// Mitsubishi GX Works2 project: BookEX2_2 Conveyor   PLC: Q13UDV

TYPE cnvBlk : STRUCT
  PIDno : DINT;  (* Pid for ECS *)
  DestBlk : INT;  (* Dest Block *)
  Status : WORD;  (* control status *)
END_STRUCT END_TYPE

// global labels: Global
VAR_GLOBAL
  gCnvBuff : ARRAY [0..19] OF cnvBlk;  (* D100~  size:4x20 = 80 word *)
  gbBlkFinish : ARRAY [0..19] OF BOOL;
  gbBlkSen : ARRAY [0..19] OF BOOL;
  gbBlkSenOn : ARRAY [0..19] OF BOOL;
  gbBlkSenOff : ARRAY [0..19] OF BOOL;
  gbBlkUp : ARRAY [0..19] OF BOOL;
  gbBlkDw : ARRAY [0..19] OF BOOL;
  gbBlkTO : ARRAY [0..19] OF BOOL;
  gbBlkTrip : ARRAY [0..19] OF BOOL;
  gbBlkData : ARRAY [0..19] OF BOOL;
  gbBlkRun : ARRAY [0..19] OF BOOL;
  gbBlkRun2 : ARRAY [0..19] OF BOOL;
  gbBlkRunUp : ARRAY [0..19] OF BOOL;
  gbBlkRunDw : ARRAY [0..19] OF BOOL;
  gbBlkRunOk : ARRAY [0..19] OF BOOL;
  gbBlkRunOk2 : ARRAY [0..19] OF BOOL;
  gbBlkEnterOk : ARRAY [0..19] OF BOOL;
END_VAR
VAR_GLOBAL CONSTANT
  cOnTime : TIME := T#300ms;
END_VAR
VAR_GLOBAL
  swOPAuto : BOOL;
  swOPEmrg : BOOL;
  gbBlkColl : BOOL;
  swNormal : BOOL;
END_VAR
VAR_GLOBAL CONSTANT
  cMaxBlk : INT := 19;
END_VAR
VAR_GLOBAL
  gwTemp AT D100 : WORD;
END_VAR
VAR_GLOBAL CONSTANT
  cMaxTime : TIME := T#15s;
  cSimTime : TIME := T#5s;
END_VAR
VAR_GLOBAL
  man01 : BOOL;
  man02 : BOOL;
  man03 : BOOL;
  man04 : BOOL;
  man05 : BOOL;
  man06 : BOOL;
  man07 : BOOL;
  man08 : BOOL;
  man09 : BOOL;
  man10 : BOOL;
  man11 : BOOL;
  man02E : BOOL;
  man05E : BOOL;
  man09E : BOOL;
  man12 : BOOL;
  man13 : BOOL;
  man12E : BOOL;
  man02Up : BOOL;
  man02Dw : BOOL;
  man05Up : BOOL;
  man05Dw : BOOL;
  man09Up : BOOL;
  man09Dw : BOOL;
  man12Up : BOOL;
  man12Dw : BOOL;
END_VAR
VAR_GLOBAL CONSTANT
  cOffTime : TIME := T#300ms;
END_VAR
VAR_GLOBAL
  swJobCmd : BOOL;
  swJobDel : BOOL;
  xSen01 AT X120 : BOOL;
  xSen02 AT X121 : BOOL;
  xSen03 AT X122 : BOOL;
  xSen04 AT X140 : BOOL;
  xSen05 AT X141 : BOOL;
  xSen06 AT X142 : BOOL;
  xSen07 AT X160 : BOOL;
  xSen08 AT X161 : BOOL;
  xSen09 AT X162 : BOOL;
  xSen10 AT X180 : BOOL;
  xSen11 AT X181 : BOOL;
  xSen12 AT X1A0 : BOOL;
  xSen13 AT X1A1 : BOOL;
  xUp02 AT X126 : BOOL;
  xDw02 AT X127 : BOOL;
  xUp05 AT X146 : BOOL;
  xDw05 AT X147 : BOOL;
  xUp09 AT X185 : BOOL;
  xDw09 AT X186 : BOOL;
  xUp12 AT X1A6 : BOOL;
  xDw12 AT X1A7 : BOOL;
  giStart AT D50 : INT;
  giEnd AT D51 : INT;
  gdPID AT D52 : DINT;
  giDel AT D54 : INT;
END_VAR
VAR_GLOBAL CONSTANT
  cSimSTime : TIME := T#2s;
END_VAR
// user libraries (not included): HMI

FUNCTION_BLOCK BlkMove
VAR_INPUT
  iCurr : INT;
  iNext : INT;
END_VAR
VAR_OUTPUT
  bRun : BOOL;
END_VAR
VAR
  idxC : INT;
  idxN : INT;
  fbTimeout : TON;
  bLoad : BOOL;
END_VAR
VAR_INPUT
  bManSw : BOOL;
END_VAR
VAR
  idxD : INT;
  fbOndelay : TON;
  fbTOdelay : TON;
  fbOffdelay : TOF;
END_VAR
VAR_INPUT
  bCurrOK : BOOL;
  bNextOK : BOOL;
END_VAR
VAR_IN_OUT
  bSimC : BOOL;
  bSimN : BOOL;
END_VAR
VAR
  fbSimCdelay : TON;
  fbSimNdelay : TON;
  bSimMode : BOOL;
  bComp : BOOL;
END_VAR
;
IF iCurr > cMaxBlk OR iCurr = 0 OR  iNext > cMaxBlk OR  iNext = 0 THEN
	bRun 	:= FALSE;
	RETURN;
END_IF;

idxC 	:= iCurr;
idxN 	:= iNext;
fbOndelay(IN:=gbBlkSen[idxC], PT:=cOnTime);			 
gbBlkSenOn[idxC] := fbOndelay.Q;
fbOffdelay(IN:= NOT gbBlkSen[idxC], PT:=cOffTime);		 
gbBlkSenOff[idxC] := fbOffdelay.Q;

(* 진입가능 검사 *)
bLoad := gbBlkSenOn[idxC] AND gbBlkData[idxC] AND NOT gbBlkFinish[idxC] AND NOT gbBlkSen[idxN] AND NOT gbBlkData[idxN] AND swOPAuto;
gbBlkEnterOk[idxN] := (gbBlkEnterOk[idxN] OR bLoad) AND NOT gbBlkSenOn[idxN] AND NOT swOPEmrg;
IF swOPAuto THEN
	bRun := ((gbBlkEnterOk[idxC] AND NOT gbBlkTO[idxC] AND bCurrOK) OR (gbBlkEnterOk[idxN] AND NOT gbBlkTO[idxN] AND bNextOK)) AND NOT swOPEmrg; 
	fbTOdelay(IN:=bRun, PT:=cMaxTime);					 
	IF fbTOdelay.Q THEN
		gbBlkTO[idxC] := TRUE;
		bRun 	:= FALSE;
	END_IF;
ELSE
	bRun := bManSw AND NOT swOPEmrg;
END_IF;

(* 시뮬레이션 동작 *)
bSimMode := NOT swNormal AND swOPAuto AND NOT swOPEmrg;
IF bSimMode THEN
	IF bRun THEN
		fbSimCdelay(IN:=gbBlkData[idxC], PT:=cSimTime);				 
		IF fbSimCdelay.Q THEN
			bSimC := FALSE;
			fbSimNdelay(IN:=gbBlkRun[idxC], PT:=cSimSTime);
			IF fbSimNdelay.Q THEN
				bSimN := TRUE;
				gCnvBuff[idxN].DestBlk 		:= gCnvBuff[idxC].DestBlk;
				gCnvBuff[idxN].PIDno		:= gCnvBuff[idxC].PIDno;
				gCnvBuff[idxC].DestBlk 		:= 0;
				gCnvBuff[idxC].PIDno		:= 0;
				gbBlkEnterOk[idxN] 			:= FALSE;
				fbSimCdelay(IN:=FALSE);
				fbSimNdelay(IN:=FALSE);
			END_IF;
		END_IF;
	ELSE
		bSimC := gbBlkData[idxC]; 
	END_IF;
ELSE
	bComp :=  gbBlkData[idxC] AND bRun AND  NOT gbBlkData[idxN] AND gbBlkSenOff[idxC] AND gbBlkSenOn[idxN];
	IF bComp THEN
		gCnvBuff[idxN].DestBlk 			:= gCnvBuff[idxC].DestBlk;
		gCnvBuff[idxN].PIDno			:= gCnvBuff[idxC].PIDno;
		gCnvBuff[idxC].DestBlk 			:= 0;
		gCnvBuff[idxC].PIDno			:= 0;
		gbBlkEnterOk[idxN] 				:= FALSE;
	END_IF;
END_IF;
END_FUNCTION_BLOCK

FUNCTION_BLOCK BlkMove2
VAR_INPUT
  iCurr : INT;
  iNext : INT;
END_VAR
VAR_OUTPUT
  bRun : BOOL;
END_VAR
VAR
  idxC : INT;
  idxN : INT;
  fbTimeout : TON;
  bLoad : BOOL;
END_VAR
VAR_INPUT
  bManSw : BOOL;
END_VAR
VAR
  idxD : INT;
  fbOndelay : TON;
  fbTOdelay : TON;
  fbOffdelay : TOF;
END_VAR
VAR_INPUT
  bCurrOK : BOOL;
  bNextOK : BOOL;
END_VAR
VAR_IN_OUT
  bSimC : BOOL;
  bSimN : BOOL;
END_VAR
VAR
  fbSimCdelay : TON;
  fbSimNdelay : TON;
  bSimMode : BOOL;
  bComp : BOOL;
END_VAR
VAR_INPUT
  bManSw2 : BOOL;
  bManUp : BOOL;
  bManDw : BOOL;
END_VAR
VAR_IN_OUT
  bSimUp : BOOL;
  bSimDw : BOOL;
END_VAR
VAR_OUTPUT
  bRun2 : BOOL;
END_VAR
VAR
  fbSimUdelay : TON;
  fbSimDdelay : TON;
  bUpCond : BOOL;
  bDwCond : BOOL;
  bTmp1 : BOOL;
  bTmp2 : BOOL;
  bTmp3 : BOOL;
  bTmp4 : BOOL;
END_VAR
;
IF iCurr > cMaxBlk OR iCurr = 0 OR  iNext > cMaxBlk OR  iNext = 0 THEN
	bRun 	:= FALSE;
	RETURN;
END_IF;

idxC 	:= iCurr;
idxN 	:= iNext;
fbOndelay(IN:=gbBlkSen[idxC], PT:=cOnTime);				 
gbBlkSenOn[idxC] := fbOndelay.Q;
fbOffdelay(IN:= NOT gbBlkSen[idxC], PT:=cOffTime);		 
gbBlkSenOff[idxC] := fbOffdelay.Q;

(* 진입가능 검사 *)
bLoad := gbBlkSenOn[idxC] AND gbBlkData[idxC] AND NOT gbBlkFinish[idxC] AND NOT gbBlkSen[idxN] AND NOT gbBlkData[idxN] AND swOPAuto;
gbBlkEnterOk[idxN] := (gbBlkEnterOk[idxN] OR bLoad) AND NOT gbBlkSenOn[idxN] AND NOT swOPEmrg;
IF swOPAuto THEN
	bRun 		:= gbBlkEnterOk[idxC] AND NOT gbBlkTO[idxC] AND bCurrOK AND NOT gbBlkFinish[idxC] AND NOT swOPEmrg;
	bRun2 	:= gbBlkEnterOk[idxN] AND NOT gbBlkTO[idxN] AND bNextOK AND NOT swOPEmrg;
	fbTOdelay(IN:=bRun OR bRun2, PT:=cMaxTime);							 
	IF fbTOdelay.Q THEN
		gbBlkTO[idxC] := TRUE;
		bRun 	:= FALSE;
	END_IF;
 	bUpCond := (gbBlkSenOn[idxC] OR gbBlkRunUp[idxC]) AND gbBlkData[idxC] AND NOT gbBlkRun[idxC] AND NOT gbBlkRun2[idxC];
	bDwCond := (gbBlkSenOff[idxC] OR gbBlkRunDw[idxC]) AND NOT gbBlkData[idxC] AND NOT gbBlkRun[idxC] AND NOT gbBlkRun2[idxC];
 	gbBlkRunUp[idxC] := bUpCond AND NOT gbBlkUp[idxC];
	gbBlkRunDw[idxC] := bDwCond AND NOT gbBlkDw[idxC];  
ELSE
	bRun := bManSw AND gbBlkDw[idxC]  AND NOT swOPEmrg;
	bRun2 := bManSw2 AND gbBlkUp[idxC] AND NOT swOPEmrg;
	gbBlkRunUp[idxC] := bManUp AND NOT gbBlkUp[idxC] AND NOT swOPEmrg;
	gbBlkRunDw[idxC] := bManDw AND NOT gbBlkDw[idxC] AND NOT swOPEmrg;
END_IF;
 
(* 시뮬레이션 동작 *)
bSimMode := NOT swNormal AND swOPAuto AND NOT swOPEmrg;
IF bSimMode THEN
	IF bRun2 THEN
		fbSimCdelay(IN:=gbBlkData[idxC], PT:=cSimSTime);	 
		IF fbSimCdelay.Q THEN
			bSimC := FALSE;
			fbSimNdelay(IN:=gbBlkRun2[idxC], PT:=cSimTime);
			IF fbSimNdelay.Q THEN
				bSimN := TRUE;
				gCnvBuff[idxN].DestBlk 		:= gCnvBuff[idxC].DestBlk;
				gCnvBuff[idxN].PIDno			:= gCnvBuff[idxC].PIDno;
				gCnvBuff[idxC].DestBlk 		:= 0;
				gCnvBuff[idxC].PIDno			:= 0;
				gbBlkEnterOk[idxN] 			:= FALSE;
				fbSimCdelay(IN:=FALSE);
				fbSimNdelay(IN:=FALSE);
			END_IF;
		END_IF;
	ELSE
		bSimC := gbBlkData[idxC]; 
	END_IF;
ELSE
	bComp :=  gbBlkData[idxC] AND bRun2 AND  NOT gbBlkData[idxN] AND gbBlkSenOff[idxC] AND gbBlkSenOn[idxN];
	IF bComp THEN
		gCnvBuff[idxN].DestBlk 			:= gCnvBuff[idxC].DestBlk;
		gCnvBuff[idxN].PIDno			:= gCnvBuff[idxC].PIDno;
		gCnvBuff[idxC].DestBlk 			:= 0;
		gCnvBuff[idxC].PIDno			:= 0;
		gbBlkEnterOk[idxN] 				:= FALSE;
	END_IF;
END_IF;

IF NOT swNormal THEN
 	fbSimUdelay(IN:=gbBlkRunUp[idxC], PT:=cSimSTime);	 
	IF fbSimUdelay.Q THEN
		bSimUp := TRUE;
		bSimDw := FALSE;
	END_IF;
	fbSimDdelay(IN:=gbBlkRunDw[idxC], PT:=cSimSTime);			 
	IF fbSimDdelay.Q THEN
		bSimUp := FALSE;
		bSimDw := TRUE;
	END_IF;
END_IF;
END_FUNCTION_BLOCK

FUNCTION_BLOCK BlkStatus
VAR_INPUT
  iEnd : INT;
  iStart : INT;
END_VAR
VAR
  idx : INT;
  wTemp : WORD;
END_VAR

FOR idx := iStart TO iEnd DO 
	wTemp := 0;		(* initialize bit *)
	gbBlkData[idx] := FALSE;
	gbBlkFinish[idx] := FALSE;
	IF gCnvBuff[idx].DestBlk <> 0 THEN
		gbBlkData[idx] := TRUE;
		IF (gCnvBuff[idx].DestBlk = idx) THEN
			gbBlkFinish[idx] := TRUE;
		END_IF;
	END_IF;
	IF gbBlkSen[idx] 		THEN	BSET(TRUE, 0, wTemp ); 		END_IF;		 
	IF gbBlkRun[idx] 		THEN	BSET(TRUE, 1, wTemp ); 		END_IF;	 
	IF gbBlkSenOn[idx] 		THEN	BSET(TRUE, 2, wTemp ); 		END_IF;			 
	IF gbBlkSenOff[idx] 	THEN	BSET(TRUE, 3, wTemp ); 		END_IF;			 
	IF gbBlkUp[idx] 		THEN	BSET(TRUE, 4, wTemp ); 		END_IF;		 	
	IF gbBlkDw[idx] 		THEN	BSET(TRUE, 5, wTemp ); 		END_IF;		 
	IF gbBlkTO[idx] 		THEN	BSET(TRUE, 6, wTemp ); 		END_IF;			 
	IF gbBlkTrip[idx] 		THEN	BSET(TRUE, 7, wTemp ); 		END_IF;		 
	IF gbBlkData[idx] 		THEN	BSET(TRUE, 8, wTemp ); 		END_IF;		 
	IF gbBlkRun2[idx] 		THEN	BSET(TRUE, 9, wTemp ); 		END_IF;			 
	IF gbBlkRunUp[idx] 		THEN	BSET(TRUE, 10, wTemp ); 	END_IF;			 
	IF gbBlkRunDw[idx] 		THEN	BSET(TRUE, 11, wTemp ); 	END_IF;			 
	IF gbBlkRunOk[idx] 		THEN	BSET(TRUE, 12, wTemp ); 	END_IF;			 
	IF gbBlkRunOk2[idx] 	THEN	BSET(TRUE, 13, wTemp ); 	END_IF;			 
	IF gbBlkFinish[idx] 	THEN	BSET(TRUE, 14, wTemp ); 	END_IF;			 
	IF gbBlkEnterOK[idx] 	THEN	BSET(TRUE, 15, wTemp ); 	END_IF;			 
	gCnvBuff[idx].Status := wTemp;
END_FOR;
END_FUNCTION_BLOCK

FUNCTION_BLOCK JobControl
VAR_INPUT
  bCmd : BOOL;
  bDel : BOOL;
  iStartBlk : INT;
  iEndBlk : INT;
  dJobPID : DINT;
  iDelBlk : INT;
END_VAR
VAR
  bOK1 : BOOL;
  bOK2 : BOOL;
END_VAR
;
bOK1 := iStartBlk > 0 AND iStartBlk <= cMaxBlk AND  iEndBlk > 0 AND iEndBlk <= cMaxBlk AND dJobPID <> 0; 
bOK2 := iDelBlk > 0 AND iDelBlk <= cMaxBlk;

IF LDP(TRUE, bCmd) AND bOK1 THEN
	gCnvBuff[iStartBlk].DestBlk := iEndBlk;
	gCnvBuff[iStartBlk].PIDno := dJobPID;	
END_IF;

IF LDP(TRUE, bDel) AND bOK2 THEN
	gCnvBuff[iDelBlk].DestBlk := 0;
	gCnvBuff[iDelBlk].PIDno := 0;
END_IF;
END_FUNCTION_BLOCK

PROGRAM ex_Ladder
(* structured ladder/FBD written out as ST: instructions are called as NAME(EN, inputs, outputs); _pN, _eN, _tN stand for wires *)
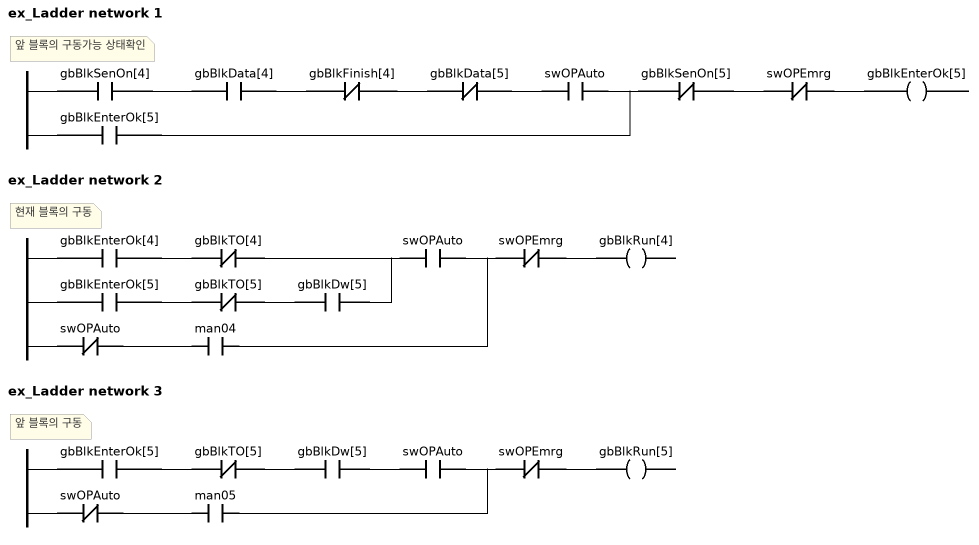
(* network 1 *)
(* 앞 블록의 구동가능 상태확인 *)
gbBlkEnterOk[5] := (((gbBlkSenOn[4] AND gbBlkData[4] AND NOT gbBlkFinish[4] AND NOT gbBlkData[5] AND swOPAuto) OR gbBlkEnterOk[5]) AND NOT gbBlkSenOn[5]) AND NOT swOPEmrg;
(* network 2 *)
(* 현재 블록의 구동 *)
gbBlkRun[4] := ((((gbBlkEnterOk[4] AND NOT gbBlkTO[4]) OR (gbBlkEnterOk[5] AND NOT gbBlkTO[5] AND gbBlkDw[5])) AND swOPAuto) OR (NOT swOPAuto AND man04)) AND NOT swOPEmrg;
(* network 3 *)
(* 앞 블록의 구동 *)
gbBlkRun[5] := ((gbBlkEnterOk[5] AND NOT gbBlkTO[5] AND gbBlkDw[5] AND swOPAuto) OR (NOT swOPAuto AND man05)) AND NOT swOPEmrg;
END_PROGRAM

PROGRAM m01_ConvIN
VAR
  Mov8BIT_1 : Mov8BIT;
  Mov8BIT_2 : Mov8BIT;
  Mov8BIT_3 : Mov8BIT;
  Mov8BIT_4 : Mov8BIT;
  Mov8BIT_5 : Mov8BIT;
  Mov8BIT_6 : Mov8BIT;
  Mov8BIT_7 : Mov8BIT;
END_VAR
(* structured ladder/FBD written out as ST: instructions are called as NAME(EN, inputs, outputs); _pN, _eN, _tN stand for wires *)
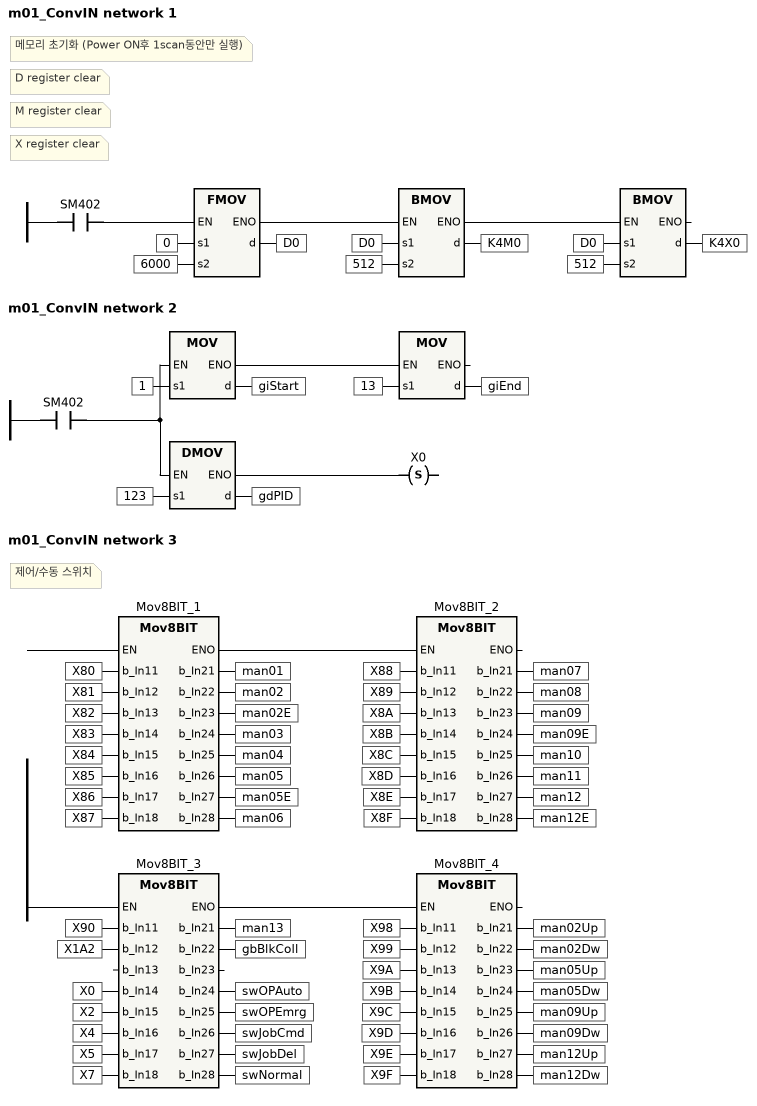
(* network 1 *)
(* 메모리 초기화 (Power ON후 1scan동안만 실행) *)
(* D register clear *)
(* M register clear *)
(* X register clear *)
_e1 := FMOV(SM402, 0, 6000, D0);
_e2 := BMOV(_e1, D0, 512, K4M0);
BMOV(_e2, D0, 512, K4X0);
(* network 2 *)
_e1 := MOV(SM402, 1, giStart);
MOV(_e1, 13, giEnd);
_e2 := DMOV(SM402, 123, gdPID);
SET(_e2, X0);
(* network 3 *)
(* 제어/수동 스위치 *)
Mov8BIT_1(EN := TRUE, b_In11 := X80, b_In12 := X81, b_In13 := X82, b_In14 := X83, b_In15 := X84, b_In16 := X85, b_In17 := X86, b_In18 := X87, b_In21 => man01, b_In22 => man02, b_In23 => man02E, b_In24 => man03, b_In25 => man04, b_In26 => man05, b_In27 => man05E, b_In28 => man06);
Mov8BIT_2(EN := Mov8BIT_1.ENO, b_In11 := X88, b_In12 := X89, b_In13 := X8A, b_In14 := X8B, b_In15 := X8C, b_In16 := X8D, b_In17 := X8E, b_In18 := X8F, b_In21 => man07, b_In22 => man08, b_In23 => man09, b_In24 => man09E, b_In25 => man10, b_In26 => man11, b_In27 => man12, b_In28 => man12E);
Mov8BIT_3(EN := TRUE, b_In11 := X90, b_In12 := X1A2, b_In14 := X0, b_In15 := X2, b_In16 := X4, b_In17 := X5, b_In18 := X7, b_In21 => man13, b_In22 => gbBlkColl, b_In24 => swOPAuto, b_In25 => swOPEmrg, b_In26 => swJobCmd, b_In27 => swJobDel, b_In28 => swNormal);
Mov8BIT_4(EN := Mov8BIT_3.ENO, b_In11 := X98, b_In12 := X99, b_In13 := X9A, b_In14 := X9B, b_In15 := X9C, b_In16 := X9D, b_In17 := X9E, b_In18 := X9F, b_In21 => man02Up, b_In22 => man02Dw, b_In23 => man05Up, b_In24 => man05Dw, b_In25 => man09Up, b_In26 => man09Dw, b_In27 => man12Up, b_In28 => man12Dw);
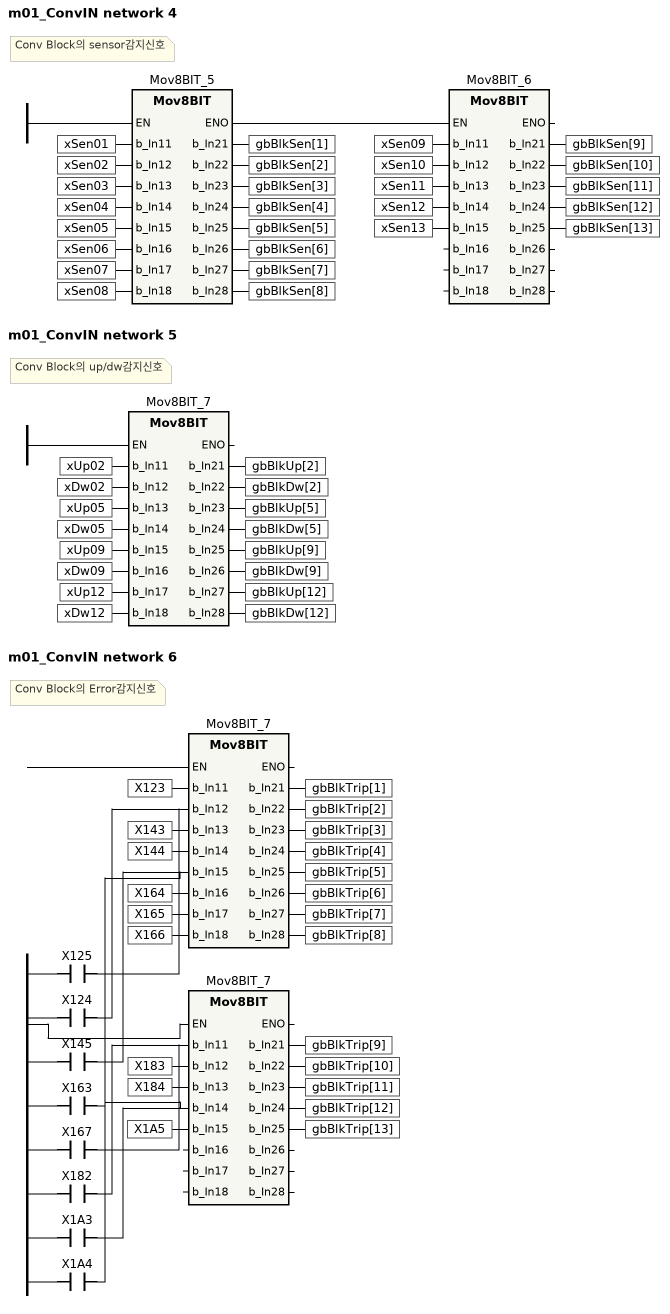
(* network 4 *)
(* Conv Block의 sensor감지신호 *)
Mov8BIT_5(EN := TRUE, b_In11 := xSen01, b_In12 := xSen02, b_In13 := xSen03, b_In14 := xSen04, b_In15 := xSen05, b_In16 := xSen06, b_In17 := xSen07, b_In18 := xSen08, b_In21 => gbBlkSen[1], b_In22 => gbBlkSen[2], b_In23 => gbBlkSen[3], b_In24 => gbBlkSen[4], b_In25 => gbBlkSen[5], b_In26 => gbBlkSen[6], b_In27 => gbBlkSen[7], b_In28 => gbBlkSen[8]);
Mov8BIT_6(EN := Mov8BIT_5.ENO, b_In11 := xSen09, b_In12 := xSen10, b_In13 := xSen11, b_In14 := xSen12, b_In15 := xSen13, b_In21 => gbBlkSen[9], b_In22 => gbBlkSen[10], b_In23 => gbBlkSen[11], b_In24 => gbBlkSen[12], b_In25 => gbBlkSen[13]);
(* network 5 *)
(* Conv Block의 up/dw감지신호 *)
Mov8BIT_7(EN := TRUE, b_In11 := xUp02, b_In12 := xDw02, b_In13 := xUp05, b_In14 := xDw05, b_In15 := xUp09, b_In16 := xDw09, b_In17 := xUp12, b_In18 := xDw12, b_In21 => gbBlkUp[2], b_In22 => gbBlkDw[2], b_In23 => gbBlkUp[5], b_In24 => gbBlkDw[5], b_In25 => gbBlkUp[9], b_In26 => gbBlkDw[9], b_In27 => gbBlkUp[12], b_In28 => gbBlkDw[12]);
(* network 6 *)
(* Conv Block의 Error감지신호 *)
Mov8BIT_7(EN := TRUE, b_In11 := X123, b_In12 := X125 OR X124, b_In13 := X143, b_In14 := X144, b_In15 := X145 OR X163, b_In16 := X164, b_In17 := X165, b_In18 := X166, b_In21 => gbBlkTrip[1], b_In22 => gbBlkTrip[2], b_In23 => gbBlkTrip[3], b_In24 => gbBlkTrip[4], b_In25 => gbBlkTrip[5], b_In26 => gbBlkTrip[6], b_In27 => gbBlkTrip[7], b_In28 => gbBlkTrip[8]);
Mov8BIT_7(EN := TRUE, b_In11 := X167 OR X182, b_In12 := X183, b_In13 := X184, b_In14 := X1A3 OR X1A4, b_In15 := X1A5, b_In21 => gbBlkTrip[9], b_In22 => gbBlkTrip[10], b_In23 => gbBlkTrip[11], b_In24 => gbBlkTrip[12], b_In25 => gbBlkTrip[13]);
END_PROGRAM

PROGRAM m02_Conveyor
VAR
  BlkMove_1 : BlkMove;
  BlkMove_7 : BlkMove;
  BlkMove_3 : BlkMove;
  BlkMove_4 : BlkMove;
  BlkMove_6 : BlkMove;
  BlkMove_8 : BlkMove;
  BlkMove_10 : BlkMove;
  BlkMove_11 : BlkMove;
  BlkMove_13 : BlkMove;
  BlkMove2_2 : BlkMove2;
  BlkMove2_5 : BlkMove2;
  BlkMove2_9 : BlkMove2;
  BlkMove2_12 : BlkMove2;
  JobControl_1 : JobControl;
  BlkStatus_1 : BlkStatus;
END_VAR
(* structured ladder/FBD written out as ST: instructions are called as NAME(EN, inputs, outputs); _pN, _eN, _tN stand for wires *)
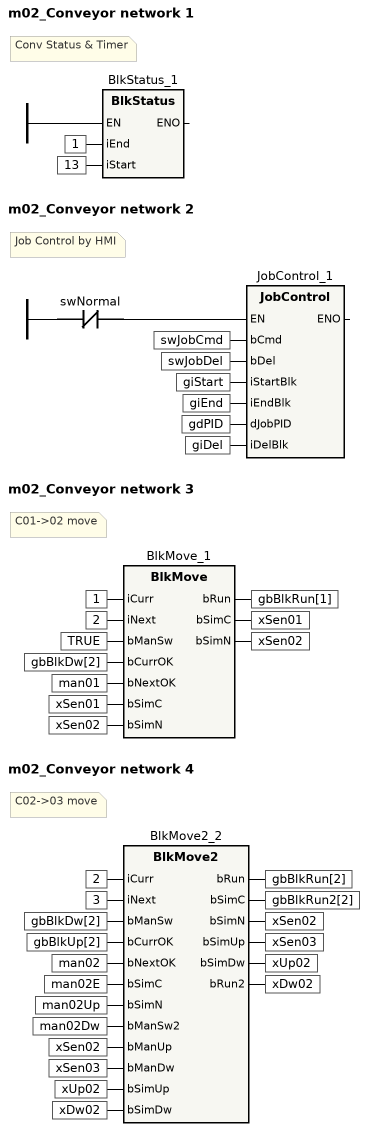
(* network 1 *)
(* Conv Status & Timer *)
BlkStatus_1(EN := TRUE, iEnd := 1, iStart := 13);
(* network 2 *)
(* Job Control by HMI *)
JobControl_1(EN := NOT swNormal, bCmd := swJobCmd, bDel := swJobDel, iStartBlk := giStart, iEndBlk := giEnd, dJobPID := gdPID, iDelBlk := giDel);
(* network 3 *)
(* C01->02 move *)
BlkMove_1(iCurr := 1, iNext := 2, bManSw := TRUE, bCurrOK := gbBlkDw[2], bNextOK := man01, bSimC := xSen01, bSimN := xSen02, bRun => gbBlkRun[1]);
xSen01 := BlkMove_1.bSimC;
xSen02 := BlkMove_1.bSimN;
(* network 4 *)
(* C02->03 move *)
BlkMove2_2(iCurr := 2, iNext := 3, bManSw := gbBlkDw[2], bCurrOK := gbBlkUp[2], bNextOK := man02, bSimC := man02E, bSimN := man02Up, bManSw2 := man02Dw, bManUp := xSen02, bManDw := xSen03, bSimUp := xUp02, bSimDw := xDw02, bRun => gbBlkRun[2], bRun2 => xDw02);
gbBlkRun2[2] := BlkMove2_2.bSimC;
xSen02 := BlkMove2_2.bSimN;
xSen03 := BlkMove2_2.bSimUp;
xUp02 := BlkMove2_2.bSimDw;
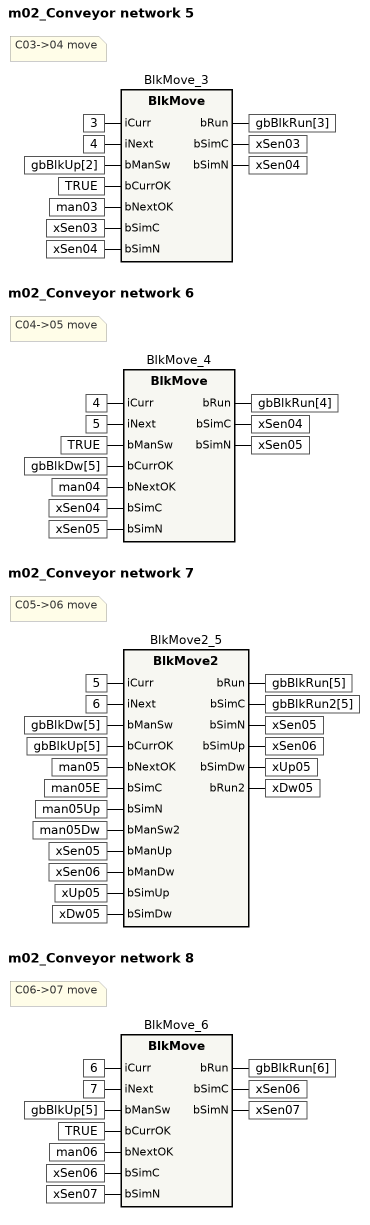
(* network 5 *)
(* C03->04 move *)
BlkMove_3(iCurr := 3, iNext := 4, bManSw := gbBlkUp[2], bCurrOK := TRUE, bNextOK := man03, bSimC := xSen03, bSimN := xSen04, bRun => gbBlkRun[3]);
xSen03 := BlkMove_3.bSimC;
xSen04 := BlkMove_3.bSimN;
(* network 6 *)
(* C04->05 move *)
BlkMove_4(iCurr := 4, iNext := 5, bManSw := TRUE, bCurrOK := gbBlkDw[5], bNextOK := man04, bSimC := xSen04, bSimN := xSen05, bRun => gbBlkRun[4]);
xSen04 := BlkMove_4.bSimC;
xSen05 := BlkMove_4.bSimN;
(* network 7 *)
(* C05->06 move *)
BlkMove2_5(iCurr := 5, iNext := 6, bManSw := gbBlkDw[5], bCurrOK := gbBlkUp[5], bNextOK := man05, bSimC := man05E, bSimN := man05Up, bManSw2 := man05Dw, bManUp := xSen05, bManDw := xSen06, bSimUp := xUp05, bSimDw := xDw05, bRun => gbBlkRun[5], bRun2 => xDw05);
gbBlkRun2[5] := BlkMove2_5.bSimC;
xSen05 := BlkMove2_5.bSimN;
xSen06 := BlkMove2_5.bSimUp;
xUp05 := BlkMove2_5.bSimDw;
(* network 8 *)
(* C06->07 move *)
BlkMove_6(iCurr := 6, iNext := 7, bManSw := gbBlkUp[5], bCurrOK := TRUE, bNextOK := man06, bSimC := xSen06, bSimN := xSen07, bRun => gbBlkRun[6]);
xSen06 := BlkMove_6.bSimC;
xSen07 := BlkMove_6.bSimN;
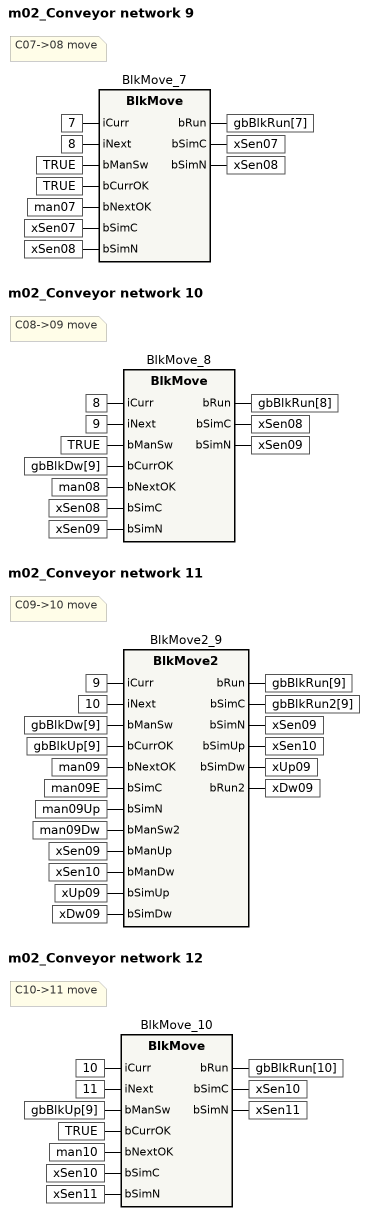
(* network 9 *)
(* C07->08 move *)
BlkMove_7(iCurr := 7, iNext := 8, bManSw := TRUE, bCurrOK := TRUE, bNextOK := man07, bSimC := xSen07, bSimN := xSen08, bRun => gbBlkRun[7]);
xSen07 := BlkMove_7.bSimC;
xSen08 := BlkMove_7.bSimN;
(* network 10 *)
(* C08->09 move *)
BlkMove_8(iCurr := 8, iNext := 9, bManSw := TRUE, bCurrOK := gbBlkDw[9], bNextOK := man08, bSimC := xSen08, bSimN := xSen09, bRun => gbBlkRun[8]);
xSen08 := BlkMove_8.bSimC;
xSen09 := BlkMove_8.bSimN;
(* network 11 *)
(* C09->10 move *)
BlkMove2_9(iCurr := 9, iNext := 10, bManSw := gbBlkDw[9], bCurrOK := gbBlkUp[9], bNextOK := man09, bSimC := man09E, bSimN := man09Up, bManSw2 := man09Dw, bManUp := xSen09, bManDw := xSen10, bSimUp := xUp09, bSimDw := xDw09, bRun => gbBlkRun[9], bRun2 => xDw09);
gbBlkRun2[9] := BlkMove2_9.bSimC;
xSen09 := BlkMove2_9.bSimN;
xSen10 := BlkMove2_9.bSimUp;
xUp09 := BlkMove2_9.bSimDw;
(* network 12 *)
(* C10->11 move *)
BlkMove_10(iCurr := 10, iNext := 11, bManSw := gbBlkUp[9], bCurrOK := TRUE, bNextOK := man10, bSimC := xSen10, bSimN := xSen11, bRun => gbBlkRun[10]);
xSen10 := BlkMove_10.bSimC;
xSen11 := BlkMove_10.bSimN;
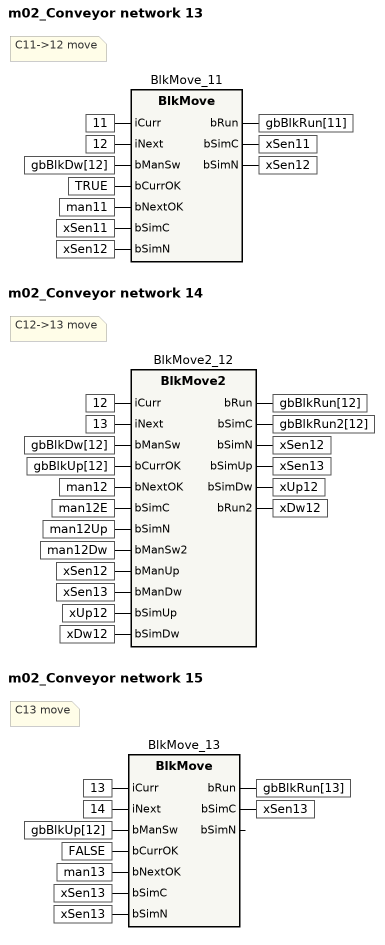
(* network 13 *)
(* C11->12 move *)
BlkMove_11(iCurr := 11, iNext := 12, bManSw := gbBlkDw[12], bCurrOK := TRUE, bNextOK := man11, bSimC := xSen11, bSimN := xSen12, bRun => gbBlkRun[11]);
xSen11 := BlkMove_11.bSimC;
xSen12 := BlkMove_11.bSimN;
(* network 14 *)
(* C12->13 move *)
BlkMove2_12(iCurr := 12, iNext := 13, bManSw := gbBlkDw[12], bCurrOK := gbBlkUp[12], bNextOK := man12, bSimC := man12E, bSimN := man12Up, bManSw2 := man12Dw, bManUp := xSen12, bManDw := xSen13, bSimUp := xUp12, bSimDw := xDw12, bRun => gbBlkRun[12], bRun2 => xDw12);
gbBlkRun2[12] := BlkMove2_12.bSimC;
xSen12 := BlkMove2_12.bSimN;
xSen13 := BlkMove2_12.bSimUp;
xUp12 := BlkMove2_12.bSimDw;
(* network 15 *)
(* C13 move *)
BlkMove_13(iCurr := 13, iNext := 14, bManSw := gbBlkUp[12], bCurrOK := FALSE, bNextOK := man13, bSimC := xSen13, bSimN := xSen13, bRun => gbBlkRun[13]);
xSen13 := BlkMove_13.bSimC;
END_PROGRAM

PROGRAM m03_ConvOUT
VAR
  Mov8BIT_1 : Mov8BIT;
  Mov8BIT_2 : Mov8BIT;
END_VAR
(* structured ladder/FBD written out as ST: instructions are called as NAME(EN, inputs, outputs); _pN, _eN, _tN stand for wires *)
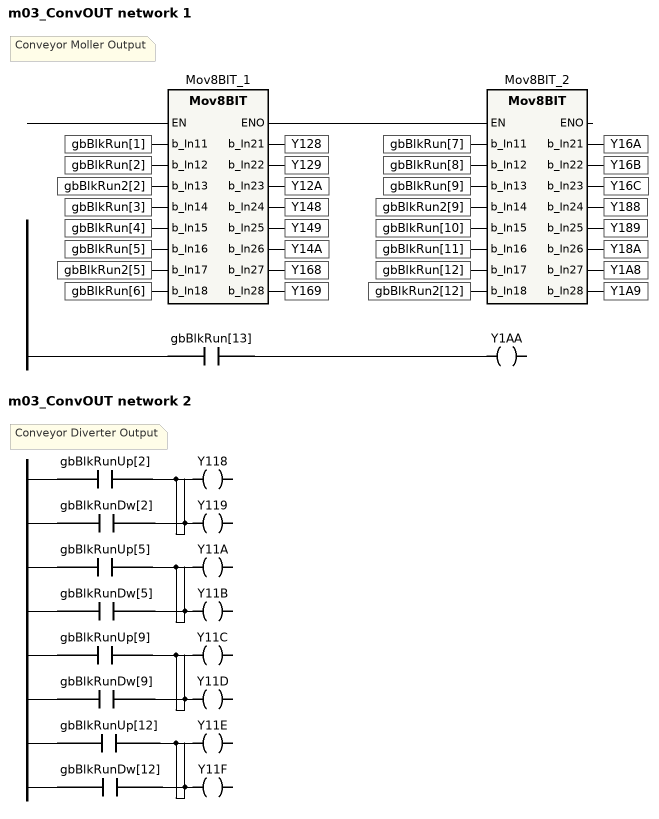
(* network 1 *)
(* Conveyor Moller Output *)
Mov8BIT_1(EN := TRUE, b_In11 := gbBlkRun[1], b_In12 := gbBlkRun[2], b_In13 := gbBlkRun2[2], b_In14 := gbBlkRun[3], b_In15 := gbBlkRun[4], b_In16 := gbBlkRun[5], b_In17 := gbBlkRun2[5], b_In18 := gbBlkRun[6], b_In21 => Y128, b_In22 => Y129, b_In23 => Y12A, b_In24 => Y148, b_In25 => Y149, b_In26 => Y14A, b_In27 => Y168, b_In28 => Y169);
Mov8BIT_2(EN := Mov8BIT_1.ENO, b_In11 := gbBlkRun[7], b_In12 := gbBlkRun[8], b_In13 := gbBlkRun[9], b_In14 := gbBlkRun2[9], b_In15 := gbBlkRun[10], b_In16 := gbBlkRun[11], b_In17 := gbBlkRun[12], b_In18 := gbBlkRun2[12], b_In21 => Y16A, b_In22 => Y16B, b_In23 => Y16C, b_In24 => Y188, b_In25 => Y189, b_In26 => Y18A, b_In27 => Y1A8, b_In28 => Y1A9);
Y1AA := gbBlkRun[13];
(* network 2 *)
(* Conveyor Diverter Output *)
_p1 := gbBlkRunUp[2] OR gbBlkRunDw[2];
Y118 := _p1;
Y119 := _p1;
_p2 := gbBlkRunUp[5] OR gbBlkRunDw[5];
Y11A := _p2;
Y11B := _p2;
_p3 := gbBlkRunUp[9] OR gbBlkRunDw[9];
Y11C := _p3;
Y11D := _p3;
_p4 := gbBlkRunUp[12] OR gbBlkRunDw[12];
Y11E := _p4;
Y11F := _p4;
END_PROGRAM
